// TIA Portal project "schody impulsowo" (V11)

(* hardware
DEVICE "S7-400 station_1"  S7400.Device
   slot 0: "UR1_0"  UR1  6ES7 400-1TA01-0AA0
   slot 2: "PLC_1"  CPU 416F-3 PN/DP  6ES7 416-3FR05-0AB0  V5.3
      slot 5: "PROFINET interface_1"  PN-IO
         slot 1: "Port_1"  Port
         slot 2: "Port_2"  Port
*)

// ===== PLC "PLC_1"  CPU 416F-3 PN/DP =====

VAR_GLOBAL   // PLC tag table "Default tag table"
   "Tag_1" AT %I0.0 : Bool;
   "Tag_2" AT %I0.1 : Bool;
   "Tag_3" AT %Q0.0 : Bool;
   "Tag_4" AT %M0.0 : Bool;
   "Tag_5" AT %M0.1 : Bool;
   "Tag_6" AT %M1.0 : Bool;
   "Tag_7" AT %M0.7 : Bool;
   "Tag_8" AT %M1.1 : Bool;
   "Tag_9" AT %M0.6 : Bool;
   "Tag_10" AT %M1.2 : Bool;
   "Tag_11" AT %M1.3 : Bool;
   "Tag_12" AT %I0.2 : Bool;
   "Tag_13" AT %M0.2 : Bool;
   "Tag_14" AT %M1.4 : Bool;
   "Tag_15" AT %M1.5 : Bool;
END_VAR

ORGANIZATION_BLOCK "Main"   // OB1, LAD
TITLE = "Main Program Sweep (Cycle)"
{ S7_Optimized_Access := 'FALSE' }
VERSION : 0.1
   VAR_TEMP
      OB1_EV_CLASS : Byte;   // Bits 0-3 = 1 (Coming event), Bits 4-7 = 1 (Event class 1)
      OB1_SCAN_1 : Byte;   // 1 (Cold restart scan 1 of OB 1), 3 (Scan 2-n of OB 1)
      OB1_PRIORITY : Byte;   // Priority of OB Execution
      OB1_OB_NUMBR : Byte;   // 1 (Organization block 1, OB1)
      OB1_RESERVED_1 : Byte;   // Reserved for system
      OB1_RESERVED_2 : Byte;   // Reserved for system
      OB1_PREV_CYCLE : Int;   // Cycle time of previous OB1 scan (milliseconds)
      OB1_MIN_CYCLE : Int;   // Minimum cycle time of OB1 (milliseconds)
      OB1_MAX_CYCLE : Int;   // Maximum cycle time of OB1 (milliseconds)
      OB1_DATE_TIME : Date_And_Time;   // Date and time OB1 started
   END_VAR
   VAR_TEMP   // added for the SCL form of the ladder/FBD networks
      _w1 : Bool;
      _w2 : Bool;
      _w3 : Bool;
      _w4 : Bool;
      _w5 : Bool;
      _w6 : Bool;
   END_VAR
BEGIN

REGION Network 1
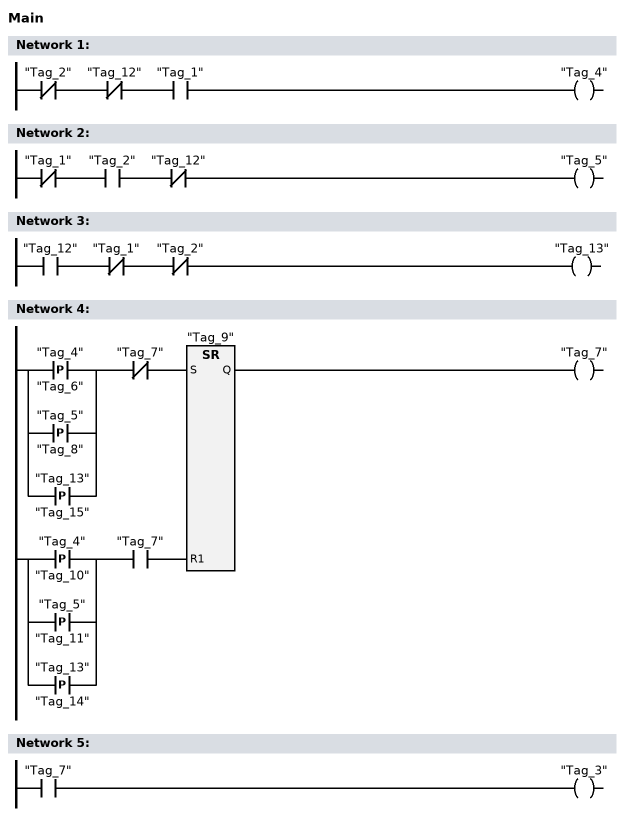
   RUNG wire#powerrail
      I_Contact( "Tag_2" )
      I_Contact( "Tag_12" )
      Contact( "Tag_1" )
      Coil( "Tag_4" )
   END_RUNG
   // the same network as SCL:
   "Tag_4" := NOT "Tag_2" AND NOT "Tag_12" AND "Tag_1";
END_REGION

REGION Network 2
   RUNG wire#powerrail
      I_Contact( "Tag_1" )
      Contact( "Tag_2" )
      I_Contact( "Tag_12" )
      Coil( "Tag_5" )
   END_RUNG
   // the same network as SCL:
   "Tag_5" := NOT "Tag_1" AND "Tag_2" AND NOT "Tag_12";
END_REGION

REGION Network 3
   RUNG wire#powerrail
      Contact( "Tag_12" )
      I_Contact( "Tag_1" )
      I_Contact( "Tag_2" )
      Coil( "Tag_13" )
   END_RUNG
   // the same network as SCL:
   "Tag_13" := "Tag_12" AND NOT "Tag_1" AND NOT "Tag_2";
END_REGION

REGION Network 4
   RUNG wire#powerrail
      P_Contact(operand := "Tag_4", bit := "Tag_6")
      wire#w1
      I_Contact( "Tag_7" )
      S_SR(operand := "Tag_9", r1 := wire#w3)
      Coil( "Tag_7" )
   END_RUNG
   RUNG wire#powerrail
      P_Contact(operand := "Tag_5", bit := "Tag_8")
   END_RUNG wire#w1
   RUNG wire#powerrail
      P_Contact(operand := "Tag_13", bit := "Tag_15")
   END_RUNG wire#w1
   RUNG wire#powerrail
      P_Contact(operand := "Tag_4", bit := "Tag_10")
      wire#w2
      Contact( "Tag_7" )
   END_RUNG wire#w3
   RUNG wire#powerrail
      P_Contact(operand := "Tag_5", bit := "Tag_11")
   END_RUNG wire#w2
   RUNG wire#powerrail
      P_Contact(operand := "Tag_13", bit := "Tag_14")
   END_RUNG wire#w2
   // the same network as SCL:
   #_w1 := "Tag_4" AND NOT "Tag_6";   // rising edge of "Tag_4"
   "Tag_6" := "Tag_4";
   #_w2 := "Tag_5" AND NOT "Tag_8";   // rising edge of "Tag_5"
   "Tag_8" := "Tag_5";
   #_w3 := "Tag_13" AND NOT "Tag_15";   // rising edge of "Tag_13"
   "Tag_15" := "Tag_13";
   #_w4 := "Tag_4" AND NOT "Tag_10";   // rising edge of "Tag_4"
   "Tag_10" := "Tag_4";
   #_w5 := "Tag_5" AND NOT "Tag_11";   // rising edge of "Tag_5"
   "Tag_11" := "Tag_5";
   #_w6 := "Tag_13" AND NOT "Tag_14";   // rising edge of "Tag_13"
   "Tag_14" := "Tag_13";
   IF (#_w1 OR #_w2 OR #_w3) AND NOT "Tag_7" THEN
       "Tag_9" := TRUE;   // SR flip-flop
   END_IF;
   IF (#_w4 OR #_w5 OR #_w6) AND "Tag_7" THEN "Tag_9" := FALSE; END_IF;
   "Tag_7" := "Tag_9";
END_REGION

REGION Network 5
   RUNG wire#powerrail
      Contact( "Tag_7" )
      Coil( "Tag_3" )
   END_RUNG
   // the same network as SCL:
   "Tag_3" := "Tag_7";
END_REGION
END_ORGANIZATION_BLOCK